FUNCTION_BLOCK FB_HeavyWash IMPLEMENTS I_WashStrategy
VAR
	   stWashSettings   : ST_WashSettings;
     bStarted   : BOOL := FALSE;
END_VAR

METHOD FB_init : BOOL
VAR_INPUT
	bInitRetains : BOOL; // if TRUE, the retain variables are initialized (warm start / cold start)
	bInCopyCode : BOOL;  // if TRUE, the instance afterwards gets moved into the copy code (online change)
END_VAR
stWashSettings.tFillDuration  := GVL_WashConstants.HEAVY_FILL;
stWashSettings.tWashDuration  := GVL_WashConstants.HEAVY_WASH;
stWashSettings.tDrainDuration := GVL_WashConstants.HEAVY_DRAIN;
stWashSettings.rWashTemperature   := GVL_WashConstants.HEAVY_TEMP;
stWashSettings.nSpinSpeed     := GVL_WashConstants.HEAVY_SPEED;
stWashSettings.sDescription   := 'Heavy wash — deep clean high temp';

FB_init := TRUE;
END_METHOD

{warning 'add method implementation '}
METHOD GetDuration : TIME
GetDuration := stWashSettings.tWashDuration;
END_METHOD

{warning 'add method implementation '}
METHOD GetProgramName : STRING
GetProgramName := 'HEAVY WASH';
END_METHOD

{warning 'add method implementation '}
METHOD GetWashSettings : ST_WashSettings
GetWashSettings := stWashSettings;
END_METHOD

{warning 'add method implementation '}
METHOD Start : BOOL
bStarted := TRUE;
Start     := TRUE;
END_METHOD

END_FUNCTION_BLOCK

(* stored: Version 1.1.0.1, ProductVersion 3.1.4024.16
   POU FB_HeavyWash: Id {7a64d12c-73d8-4e64-bb4e-97a85d4655e4}, SpecialFunc None
   Method FB_init: Id {89980812-f46a-40e8-99e6-e1e2408bf267}
   Method GetDuration: Id {dda96a2d-8014-43ae-8ba3-119d853482e1}
   Method GetProgramName: Id {0e16af83-e735-4cdc-a8a6-afe4cfcbf01e}
   Method GetWashSettings: Id {999df4b4-d99b-4e82-b5ee-689b9b37e11a}
   Method Start: Id {b7acfd0a-746c-4e30-9823-f7d32e8951b3} *)
